FUNCTION_BLOCK FB_EventFMZ
VAR_INPUT
	FB_Bacnet : FB_BACnet_DAIKIN_MasterStation_III_No_1;
END_VAR
VAR_OUTPUT
END_VAR
VAR
	fbMsg : FB_TcMessage;
	aUnits : ARRAY[1..21] OF AC_Unit_Status;
	stUnit   : AC_Unit_Status;
	i: INT;
	sMsgText: STRING;
	triggerTest : BOOL;
END_VAR
VAR RETAIN
	aPrevState : ARRAY[1..21] OF BOOL := [FALSE(*21*)];
END_VAR


aUnits[1].bPresVal := FB_Bacnet.StartStopStatus_064.bPresVal;
aUnits[1].sUnitName := 'FMZ-1 (1-00)';
aUnits[2].bPresVal := FB_Bacnet.StartStopStatus_065.bPresVal;
aUnits[2].sUnitName := 'FMZ-2 (1-01)';
aUnits[3].bPresVal := FB_Bacnet.StartStopStatus_066.bPresVal;
aUnits[3].sUnitName := 'FMZ-3 (1-02)';
aUnits[4].bPresVal := FB_Bacnet.StartStopStatus_067.bPresVal;
aUnits[4].sUnitName := 'FMZ-4 (1-03)';
aUnits[5].bPresVal := FB_Bacnet.StartStopStatus_068.bPresVal;
aUnits[5].sUnitName := 'FMZ-5 (1-04)';
aUnits[6].bPresVal := FB_Bacnet.StartStopStatus_069.bPresVal;
aUnits[6].sUnitName := 'FMZ-6 (1-05)';
aUnits[7].bPresVal := FB_Bacnet.StartStopStatus_070.bPresVal;
aUnits[7].sUnitName := 'FMZ-7 (1-06)';
aUnits[8].bPresVal := FB_Bacnet.StartStopStatus_071.bPresVal;
aUnits[8].sUnitName := 'FMZ-8 (1-07)';
aUnits[9].bPresVal := FB_Bacnet.StartStopStatus_072.bPresVal;
aUnits[9].sUnitName := 'FMZ-9 (1-08)';
aUnits[10].bPresVal := FB_Bacnet.StartStopStatus_073.bPresVal;
aUnits[10].sUnitName := 'FMZ-10 (1-09)';
aUnits[11].bPresVal := FB_Bacnet.StartStopStatus_074.bPresVal;
aUnits[11].sUnitName := 'FMZ-11 (1-10)';
aUnits[12].bPresVal := FB_Bacnet.StartStopStatus_075.bPresVal;
aUnits[12].sUnitName := 'FMZ-12 (1-11)';
aUnits[13].bPresVal := FB_Bacnet.StartStopStatus_076.bPresVal;
aUnits[13].sUnitName := 'FMZ-13 (1-12)';
aUnits[14].bPresVal := FB_Bacnet.StartStopStatus_077.bPresVal;
aUnits[14].sUnitName := 'FMZ-14 (1-13)';
aUnits[15].bPresVal := FB_Bacnet.StartStopStatus_078.bPresVal;
aUnits[15].sUnitName := 'FMZ-15 (1-14)';
aUnits[16].bPresVal := FB_Bacnet.StartStopStatus_079.bPresVal;
aUnits[16].sUnitName := 'FMZ-16 (1-15)';
aUnits[17].bPresVal := FB_Bacnet.StartStopStatus_080.bPresVal;
aUnits[17].sUnitName := 'FMZ-17 (2-00)';
aUnits[18].bPresVal := FB_Bacnet.StartStopStatus_081.bPresVal;
aUnits[18].sUnitName := 'FMZ-18 (2-01)';
aUnits[19].bPresVal := FB_Bacnet.StartStopStatus_082.bPresVal;
aUnits[19].sUnitName := 'FMZ-19 (2-02)';
aUnits[20].bPresVal := FB_Bacnet.StartStopStatus_083.bPresVal;
aUnits[20].sUnitName := 'FMZ-20 (2-03)';
aUnits[21].bPresVal := FB_Bacnet.StartStopStatus_084.bPresVal;
aUnits[21].sUnitName := 'FMZ-21 (2-04)';

FOR i := 1 TO 21 DO
	stUnit := aUnits[i]; // extract the structure instance
    IF aUnits[i].bPresVal <> aPrevState[i] THEN
        IF aUnits[i].bPresVal THEN
            sMsgText := CONCAT(stUnit.sUnitName, ' is Turned ON');
        ELSE
            sMsgText := CONCAT(stUnit.sUnitName, ' is Turned OFF');
        END_IF
		fbMsg.CreateEx(TC_EVENTS.UnitPowerStatus.EventPowerStatus, 0);
		fbMsg.ipArguments.AddString(sMsgText);
		fbMsg.Send(0);
		
        // Update previous state
        aPrevState[i] := aUnits[i].bPresVal;
    END_IF
END_FOR

END_FUNCTION_BLOCK

(* stored: Version 1.1.0.1, ProductVersion 3.1.4024.14
   POU FB_EventFMZ: Id {4f82fc44-513c-4e88-8ff0-0f3a524deed5}, SpecialFunc None *)
